SYSTEM LIFTER_MVCDL (* Lifter Control+Diagnostics with Feed & Takeoff Conveyors *)
  (* Standard: 61499-1; Classification: Simulation; ApplicationDomain: Assembly; Type: Dual Stroke Cylinder *)
  (* Version 0.5, 2008-02-18, JHC, Holobloc Inc, Added init delay to DIAGNOSTICS.LOG *)
  (* Version 0.4, 2007-11-08, JHC, Holobloc Inc, Changed device order: DIAGNOSTICS, MODEL, CONTROL. *)
  (* Version 0.3, 2007-07-08, JHC, Holobloc Inc, Added MODEL.CLOCK.CLK_DLY. *)
  (* Version 0.2, 2004-12-19, JHC, Rockwell Automation, Adjusted frame heights for WinXP. *)
  (* Version 0.1, 2004-11-12, JHC, Rockwell Automation, Combined XFER_MDL+FLT_MDL as in LIFTER_MVCL. *)
  (* Version 0.0, 2004-11-10, JHC, Rockwell Automation, Extended from LIFTER_MVCL. *)
  DEVICE DIAGNOSTICS : FRAME_DEVICE(BOUNDS := [100,360,485,150], GRID := [1,1])
    RESOURCE LOG : PANEL_RESOURCE(ROWS := 1, COLS := 1)
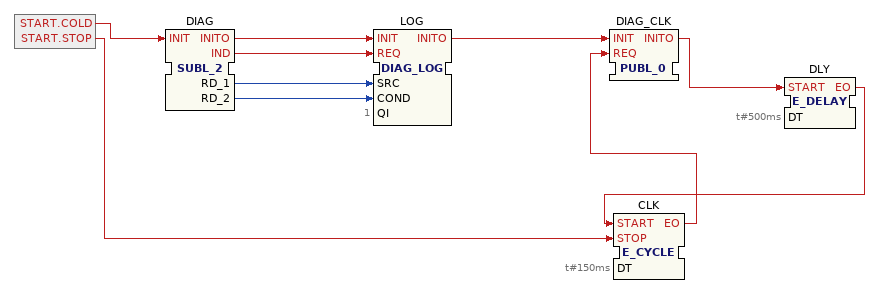
      FBS
        DIAG : SUBL_2;
        LOG : DIAG_LOG(QI := 1);
        CLK : E_CYCLE(DT := t#150ms);
        DIAG_CLK : PUBL_0;
        DLY : E_DELAY(DT := t#500ms);
      END_FBS
      EVENT_CONNECTIONS
        START.COLD TO DIAG.INIT;
        DIAG.INITO TO LOG.INIT;
        DIAG.IND TO LOG.REQ;
        LOG.INITO TO DIAG_CLK.INIT;
        CLK.EO TO DIAG_CLK.REQ;
        DIAG_CLK.INITO TO DLY.START;
        DLY.EO TO CLK.START;
        START.STOP TO CLK.STOP;
      END_CONNECTIONS
      DATA_CONNECTIONS
        DIAG.RD_1 TO LOG.SRC;
        DIAG.RD_2 TO LOG.COND;
      END_CONNECTIONS
    END_RESOURCE
    RESOURCE MONITOR : EMB_RES
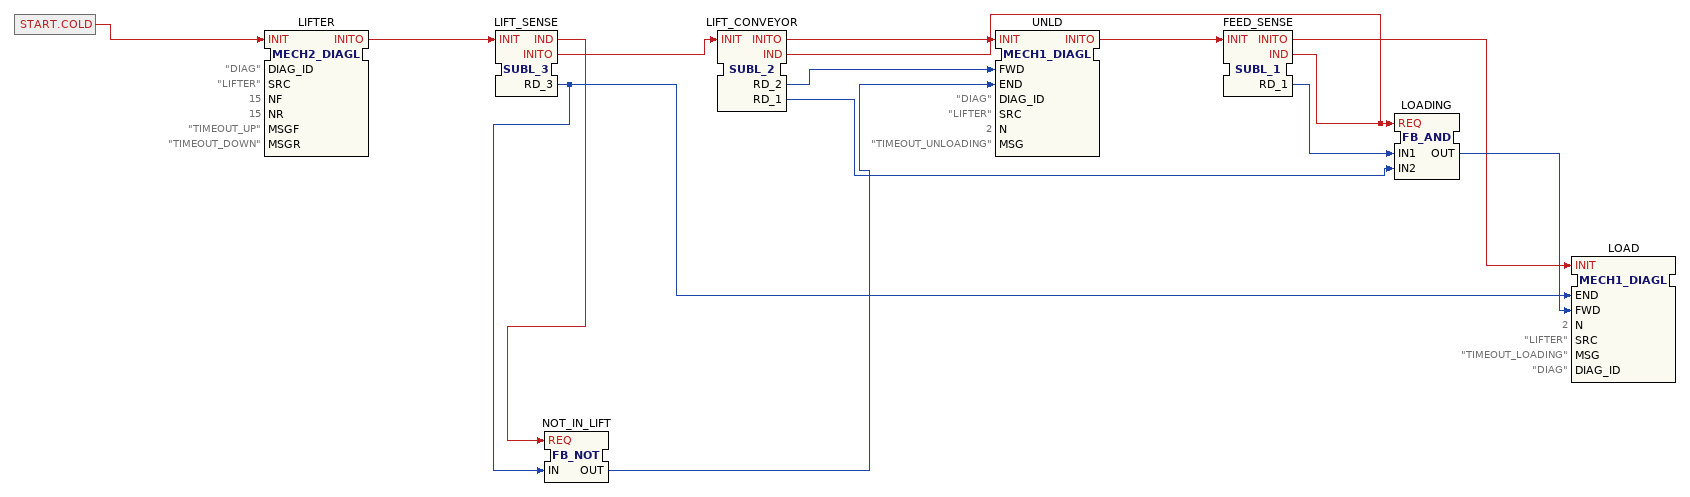
      FBS
        LIFTER : MECH2_DIAGL(DIAG_ID := "DIAG", SRC := "LIFTER", NF := 15, NR := 15, MSGF := "TIMEOUT_UP", MSGR := "TIMEOUT_DOWN");
        UNLD : MECH1_DIAGL(DIAG_ID := "DIAG", SRC := "LIFTER", N := 2, MSG := "TIMEOUT_UNLOADING"); (* Monitor Lift Unloading *)
        LIFT_CONVEYOR : SUBL_2;
        LIFT_SENSE : SUBL_3;
        NOT_IN_LIFT : FB_NOT;
        LOAD : MECH1_DIAGL(N := 2, SRC := "LIFTER", MSG := "TIMEOUT_LOADING", DIAG_ID := "DIAG");
        FEED_SENSE : SUBL_1;
        LOADING : FB_AND;
      END_FBS
      EVENT_CONNECTIONS
        START.COLD TO LIFTER.INIT;
        LIFT_SENSE.IND TO NOT_IN_LIFT.REQ;
        LIFTER.INITO TO LIFT_SENSE.INIT;
        LIFT_SENSE.INITO TO LIFT_CONVEYOR.INIT;
        LIFT_CONVEYOR.INITO TO UNLD.INIT;
        UNLD.INITO TO FEED_SENSE.INIT;
        FEED_SENSE.INITO TO LOAD.INIT;
        FEED_SENSE.IND TO LOADING.REQ;
        LIFT_CONVEYOR.IND TO LOADING.REQ;
      END_CONNECTIONS
      DATA_CONNECTIONS
        LIFT_CONVEYOR.RD_2 TO UNLD.FWD;
        NOT_IN_LIFT.OUT TO UNLD.END;
        LIFT_SENSE.RD_3 TO NOT_IN_LIFT.IN;
        LIFT_SENSE.RD_3 TO LOAD.END;
        LOADING.OUT TO LOAD.FWD;
        FEED_SENSE.RD_1 TO LOADING.IN1;
        LIFT_CONVEYOR.RD_1 TO LOADING.IN2;
      END_CONNECTIONS
    END_RESOURCE
  END_DEVICE
  DEVICE MODEL : FRAME_DEVICE(BOUNDS := [425,100,160,260])
    RESOURCE CLOCK : EMB_RES
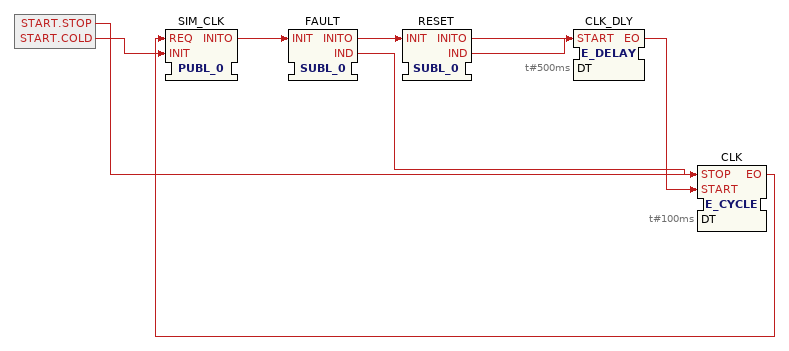
      FBS
        CLK : E_CYCLE(DT := t#100ms);
        SIM_CLK : PUBL_0;
        FAULT : SUBL_0;
        RESET : SUBL_0;
        CLK_DLY : E_DELAY(DT := t#500ms);
      END_FBS
      EVENT_CONNECTIONS
        START.STOP TO CLK.STOP;
        CLK.EO TO SIM_CLK.REQ;
        START.COLD TO SIM_CLK.INIT;
        SIM_CLK.INITO TO FAULT.INIT;
        FAULT.INITO TO RESET.INIT;
        FAULT.IND TO CLK.STOP;
        RESET.INITO TO CLK_DLY.START;
        RESET.IND TO CLK_DLY.START;
        CLK_DLY.EO TO CLK.START;
      END_CONNECTIONS
    END_RESOURCE
    RESOURCE FEED_MDL : EMB_RES
      FBS
        FEED : CNVG_MDLL(VF := 20, VS := 50);
        FEED_UNLD : SUBL_0;
        RESET : SUBL_0;
        WARN : SUBL_2;
        WARNING : LOADLE(LPOS := 100, STYLE := VSTYLE#PALLET, WKPC := [255,255,0], ID := "FEED_LOAD");
        JAM_OR_HALFIN : FB_OR;
        FAULT : SUBL_2;
        CRUSHED : E_PERMIT;
        DROPPED : LOADLE(ID := "FEED_LOAD", LPOS := 100, STYLE := VSTYLE#PALLET, WKPC := [255,0,0]);
      END_FBS
      EVENT_CONNECTIONS
        START.COLD TO FEED.INIT;
        FEED.INITO TO FEED_UNLD.INIT;
        FEED_UNLD.IND TO FEED.UNLD;
        FEED_UNLD.INITO TO RESET.INIT;
        RESET.IND TO FEED.UNLD;
        RESET.INITO TO WARN.INIT;
        START.COLD TO FAULT.INIT;
        WARN.INITO TO WARNING.INIT;
        JAM_OR_HALFIN.CNF TO WARNING.REQ;
        FAULT.IND TO CRUSHED.EI;
        CRUSHED.EO TO FEED.UNLD;
        FAULT.IND TO DROPPED.REQ;
        WARNING.INITO TO DROPPED.INIT;
        WARN.IND TO JAM_OR_HALFIN.REQ;
      END_CONNECTIONS
      DATA_CONNECTIONS
        WARN.RD_1 TO JAM_OR_HALFIN.IN1;
        WARN.RD_2 TO JAM_OR_HALFIN.IN2;
        JAM_OR_HALFIN.OUT TO WARNING.QI;
        FAULT.RD_1 TO CRUSHED.PERMIT;
        FAULT.RD_2 TO DROPPED.QI;
      END_CONNECTIONS
    END_RESOURCE
    RESOURCE LIFTER_MDL : EMB_RES
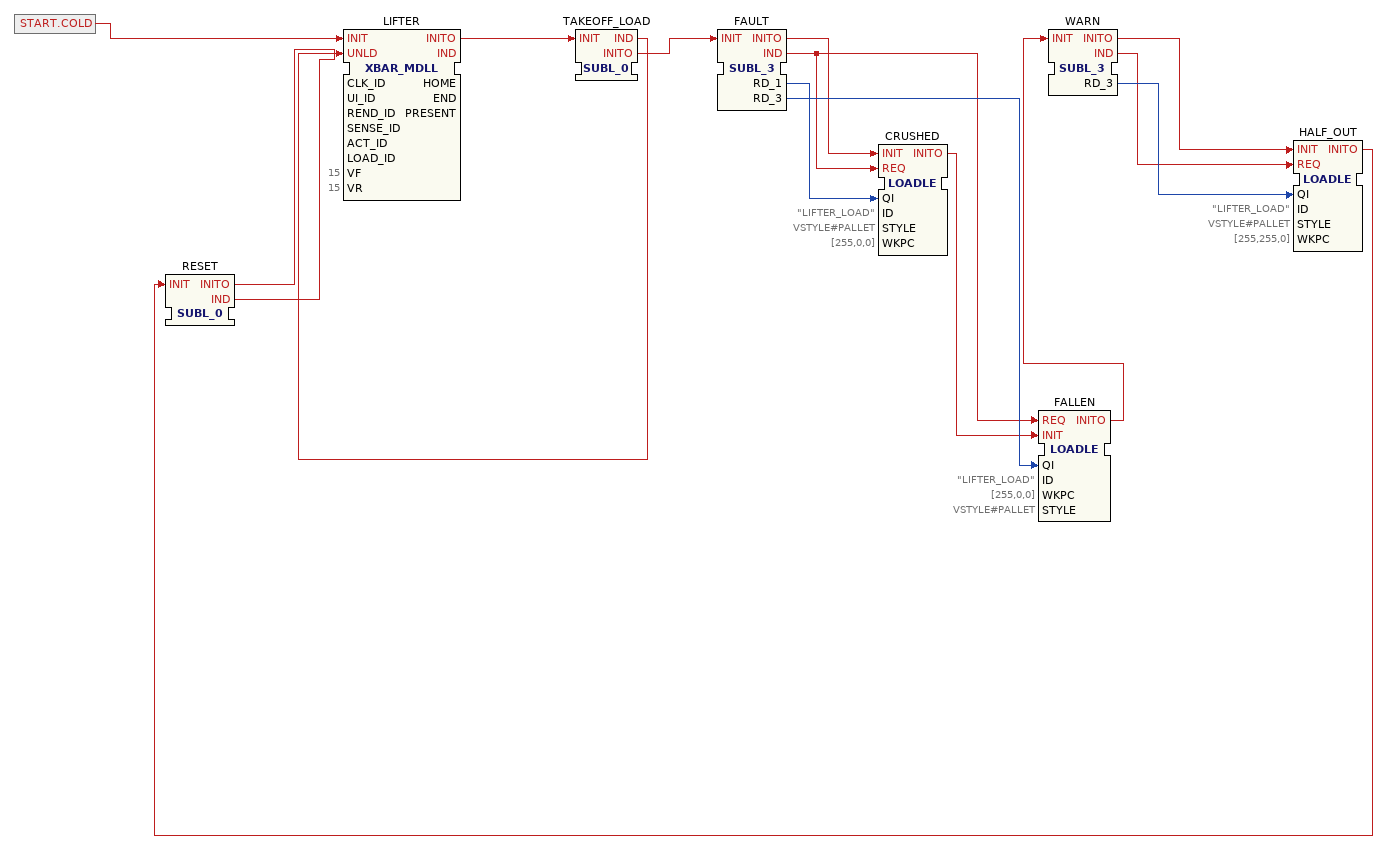
      FBS
        LIFTER : XBAR_MDLL(VF := 15, VR := 15);
        TAKEOFF_LOAD : SUBL_0;
        FAULT : SUBL_3;
        CRUSHED : LOADLE(ID := "LIFTER_LOAD", STYLE := VSTYLE#PALLET, WKPC := [255,0,0]);
        FALLEN : LOADLE(ID := "LIFTER_LOAD", WKPC := [255,0,0], STYLE := VSTYLE#PALLET);
        RESET : SUBL_0;
        WARN : SUBL_3;
        HALF_OUT : LOADLE(ID := "LIFTER_LOAD", STYLE := VSTYLE#PALLET, WKPC := [255,255,0]);
      END_FBS
      EVENT_CONNECTIONS
        START.COLD TO LIFTER.INIT;
        LIFTER.INITO TO TAKEOFF_LOAD.INIT;
        TAKEOFF_LOAD.IND TO LIFTER.UNLD;
        TAKEOFF_LOAD.INITO TO FAULT.INIT;
        FAULT.INITO TO CRUSHED.INIT;
        FAULT.IND TO CRUSHED.REQ;
        FAULT.IND TO FALLEN.REQ;
        CRUSHED.INITO TO FALLEN.INIT;
        WARN.INITO TO HALF_OUT.INIT;
        WARN.IND TO HALF_OUT.REQ;
        RESET.INITO TO LIFTER.UNLD;
        RESET.IND TO LIFTER.UNLD;
        FALLEN.INITO TO WARN.INIT;
        HALF_OUT.INITO TO RESET.INIT;
      END_CONNECTIONS
      DATA_CONNECTIONS
        FAULT.RD_1 TO CRUSHED.QI;
        FAULT.RD_3 TO FALLEN.QI;
        WARN.RD_3 TO HALF_OUT.QI;
      END_CONNECTIONS
    END_RESOURCE
    RESOURCE XFER_MDL : EMB_RES (* Pallet Transfer Model *)
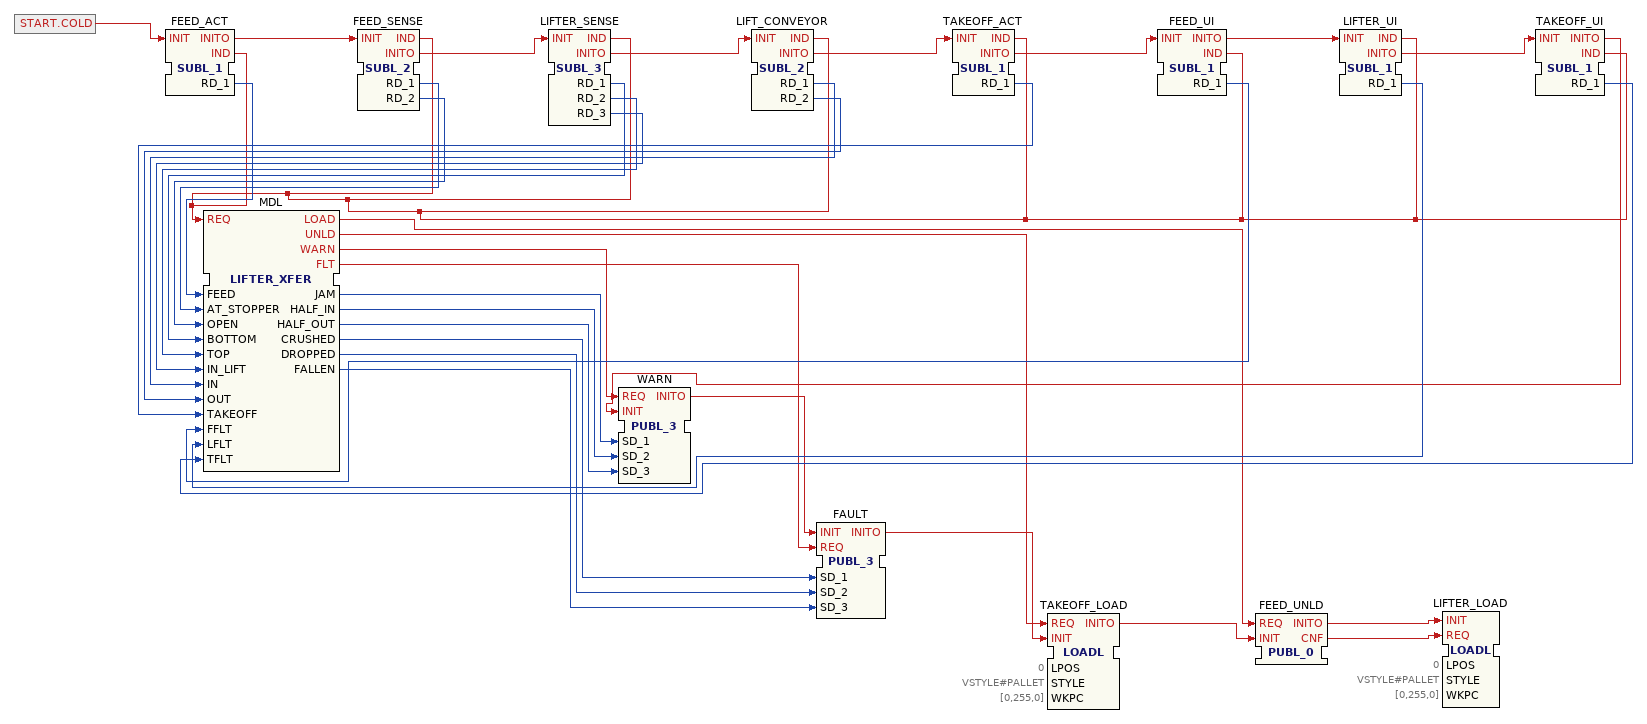
      FBS
        MDL : LIFTER_XFER;
        FEED_ACT : SUBL_1;
        FEED_SENSE : SUBL_2;
        LIFTER_SENSE : SUBL_3;
        LIFT_CONVEYOR : SUBL_2;
        TAKEOFF_ACT : SUBL_1;
        LIFTER_LOAD : LOADL(LPOS := 0, STYLE := VSTYLE#PALLET, WKPC := [0,255,0]);
        TAKEOFF_LOAD : LOADL(LPOS := 0, STYLE := VSTYLE#PALLET, WKPC := [0,255,0]);
        LIFTER_UI : SUBL_1;
        WARN : PUBL_3;
        FAULT : PUBL_3;
        FEED_UNLD : PUBL_0;
        FEED_UI : SUBL_1;
        TAKEOFF_UI : SUBL_1;
      END_FBS
      EVENT_CONNECTIONS
        START.COLD TO FEED_ACT.INIT;
        FEED_ACT.INITO TO FEED_SENSE.INIT;
        FEED_ACT.IND TO MDL.REQ;
        FEED_SENSE.IND TO MDL.REQ;
        FEED_SENSE.INITO TO LIFTER_SENSE.INIT;
        LIFTER_SENSE.IND TO MDL.REQ;
        LIFTER_SENSE.INITO TO LIFT_CONVEYOR.INIT;
        LIFT_CONVEYOR.IND TO MDL.REQ;
        LIFT_CONVEYOR.INITO TO TAKEOFF_ACT.INIT;
        TAKEOFF_ACT.IND TO MDL.REQ;
        LIFTER_UI.IND TO MDL.REQ;
        MDL.UNLD TO TAKEOFF_LOAD.REQ;
        WARN.INITO TO FAULT.INIT;
        MDL.WARN TO WARN.REQ;
        MDL.FLT TO FAULT.REQ;
        FAULT.INITO TO TAKEOFF_LOAD.INIT;
        MDL.LOAD TO FEED_UNLD.REQ;
        FEED_UNLD.INITO TO LIFTER_LOAD.INIT;
        FEED_UNLD.CNF TO LIFTER_LOAD.REQ;
        TAKEOFF_LOAD.INITO TO FEED_UNLD.INIT;
        TAKEOFF_ACT.INITO TO FEED_UI.INIT;
        FEED_UI.INITO TO LIFTER_UI.INIT;
        LIFTER_UI.INITO TO TAKEOFF_UI.INIT;
        TAKEOFF_UI.INITO TO WARN.INIT;
        FEED_UI.IND TO MDL.REQ;
        TAKEOFF_UI.IND TO MDL.REQ;
      END_CONNECTIONS
      DATA_CONNECTIONS
        FEED_ACT.RD_1 TO MDL.FEED;
        FEED_SENSE.RD_1 TO MDL.AT_STOPPER;
        LIFTER_SENSE.RD_1 TO MDL.BOTTOM;
        LIFTER_SENSE.RD_2 TO MDL.TOP;
        LIFTER_SENSE.RD_3 TO MDL.IN_LIFT;
        LIFT_CONVEYOR.RD_1 TO MDL.IN;
        LIFT_CONVEYOR.RD_2 TO MDL.OUT;
        TAKEOFF_ACT.RD_1 TO MDL.TAKEOFF;
        FEED_SENSE.RD_2 TO MDL.OPEN;
        LIFTER_UI.RD_1 TO MDL.LFLT;
        MDL.JAM TO WARN.SD_1;
        MDL.HALF_IN TO WARN.SD_2;
        MDL.HALF_OUT TO WARN.SD_3;
        MDL.CRUSHED TO FAULT.SD_1;
        MDL.DROPPED TO FAULT.SD_2;
        MDL.FALLEN TO FAULT.SD_3;
        FEED_UI.RD_1 TO MDL.FFLT;
        TAKEOFF_UI.RD_1 TO MDL.TFLT;
      END_CONNECTIONS
    END_RESOURCE
    RESOURCE TAKEOFF_MDL : EMB_RES
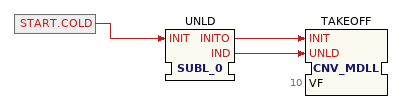
      FBS
        TAKEOFF : CNV_MDLL(VF := 10);
        UNLD : SUBL_0;
      END_FBS
      EVENT_CONNECTIONS
        START.COLD TO UNLD.INIT;
        UNLD.INITO TO TAKEOFF.INIT;
        UNLD.IND TO TAKEOFF.UNLD;
      END_CONNECTIONS
    END_RESOURCE
    RESOURCE UI : PANEL_RESOURCE(ROWS := 2, COLS := 2)
      FBS
        FAULT_IND : OUT_BOOL(LABEL := "FAULT ", C1 := [255,0,0]);
        RESET_PB : IN_EVENT(LABEL := "RESET");
        RESET : PUBL_0;
        LOAD_PB : IN_EVENT(LABEL := "LOAD");
        UNLD_PB : IN_EVENT(LABEL := "UNLOAD");
        FEED_LOAD : LOADL(STYLE := VSTYLE#PALLET, WKPC := [0,255,0]);
        UNLD : PUBL_0;
        FLT : E_RS;
        FAULT : SUBL_0;
      END_FBS
      EVENT_CONNECTIONS
        FAULT_IND.INITO TO RESET_PB.INIT;
        RESET_PB.INITO TO RESET.INIT;
        RESET_PB.IND TO RESET.REQ;
        START.COLD TO LOAD_PB.INIT;
        LOAD_PB.INITO TO FEED_LOAD.INIT;
        FEED_LOAD.INITO TO UNLD_PB.INIT;
        LOAD_PB.IND TO FEED_LOAD.REQ;
        UNLD_PB.INITO TO UNLD.INIT;
        UNLD_PB.IND TO UNLD.REQ;
        UNLD.INITO TO FAULT_IND.INIT;
        RESET.CNF TO UNLD.REQ;
        FLT.EO TO FAULT_IND.REQ;
        RESET.INITO TO FAULT.INIT;
        FAULT.IND TO FLT.S;
        UNLD.CNF TO FLT.R;
      END_CONNECTIONS
      DATA_CONNECTIONS
        FLT.Q TO FAULT_IND.IN;
      END_CONNECTIONS
    END_RESOURCE
    RESOURCE VIEW : VIEW_PANEL(DIA := 30, SIZE := [5,5], VERTICAL := 1)
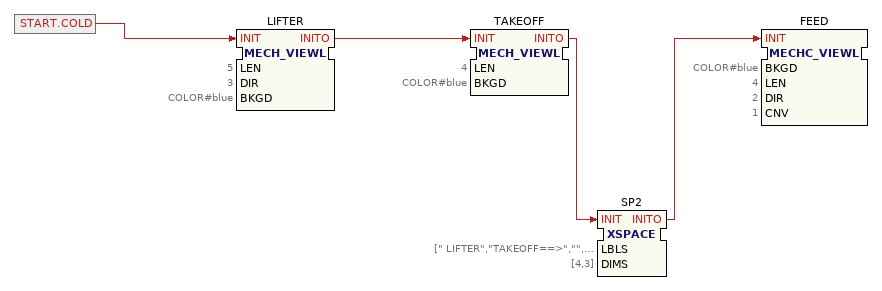
      FBS
        LIFTER : MECH_VIEWL(LEN := 5, DIR := 3, BKGD := COLOR#blue);
        FEED : MECHC_VIEWL(BKGD := COLOR#blue, LEN := 4, DIR := 2, CNV := 1); (* Feed Conveyor *)
        SP2 : XSPACE(LBLS := [" LIFTER","TAKEOFF==>","","<==FEED"], DIMS := [4,3]);
        TAKEOFF : MECH_VIEWL(LEN := 4, BKGD := COLOR#blue); (* Takeoff Conveyor *)
      END_FBS
      EVENT_CONNECTIONS
        TAKEOFF.INITO TO SP2.INIT;
        SP2.INITO TO FEED.INIT;
        START.COLD TO LIFTER.INIT;
        LIFTER.INITO TO TAKEOFF.INIT;
      END_CONNECTIONS
    END_RESOURCE
  END_DEVICE
  DEVICE CONTROL : FRAME_DEVICE(BOUNDS := [100,100,325,260], GRID := [3,2]) (* Lifter Control + HMI *)
    RESOURCE CTL : EMB_RES
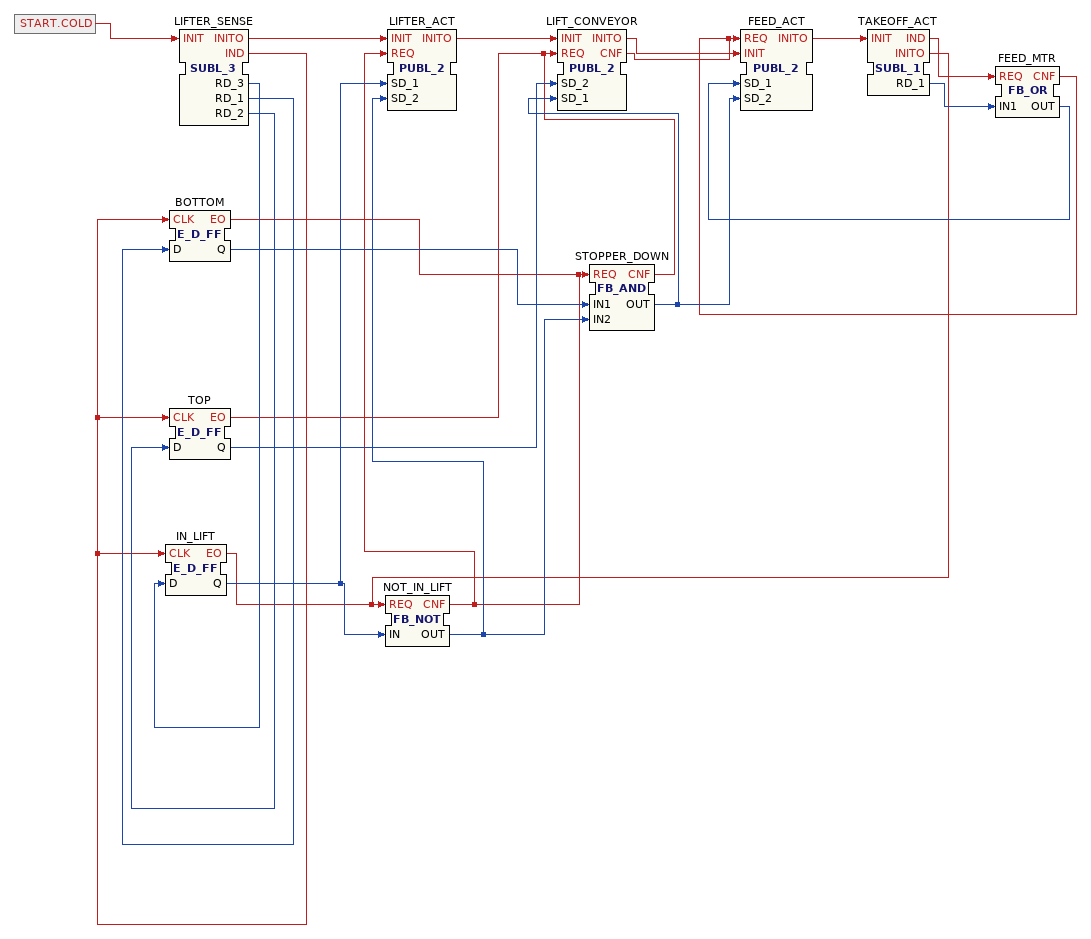
      FBS
        LIFTER_SENSE : SUBL_3;
        FEED_ACT : PUBL_2;
        LIFTER_ACT : PUBL_2;
        LIFT_CONVEYOR : PUBL_2;
        TAKEOFF_ACT : SUBL_1;
        FEED_MTR : FB_OR;
        IN_LIFT : E_D_FF;
        BOTTOM : E_D_FF;
        TOP : E_D_FF;
        NOT_IN_LIFT : FB_NOT;
        STOPPER_DOWN : FB_AND;
      END_FBS
      EVENT_CONNECTIONS
        START.COLD TO LIFTER_SENSE.INIT;
        FEED_ACT.INITO TO TAKEOFF_ACT.INIT;
        TAKEOFF_ACT.IND TO FEED_MTR.REQ;
        FEED_MTR.CNF TO FEED_ACT.REQ;
        LIFTER_SENSE.INITO TO LIFTER_ACT.INIT;
        LIFTER_ACT.INITO TO LIFT_CONVEYOR.INIT;
        LIFT_CONVEYOR.INITO TO FEED_ACT.INIT;
        LIFTER_SENSE.IND TO IN_LIFT.CLK;
        LIFTER_SENSE.IND TO TOP.CLK;
        LIFTER_SENSE.IND TO BOTTOM.CLK;
        IN_LIFT.EO TO NOT_IN_LIFT.REQ;
        NOT_IN_LIFT.CNF TO LIFTER_ACT.REQ;
        TOP.EO TO LIFT_CONVEYOR.REQ;
        BOTTOM.EO TO STOPPER_DOWN.REQ;
        NOT_IN_LIFT.CNF TO STOPPER_DOWN.REQ;
        TAKEOFF_ACT.INITO TO NOT_IN_LIFT.REQ;
        LIFT_CONVEYOR.CNF TO FEED_ACT.REQ;
        STOPPER_DOWN.CNF TO LIFT_CONVEYOR.REQ;
      END_CONNECTIONS
      DATA_CONNECTIONS
        TAKEOFF_ACT.RD_1 TO FEED_MTR.IN1;
        FEED_MTR.OUT TO FEED_ACT.SD_1;
        LIFTER_SENSE.RD_3 TO IN_LIFT.D;
        LIFTER_SENSE.RD_1 TO BOTTOM.D;
        LIFTER_SENSE.RD_2 TO TOP.D;
        IN_LIFT.Q TO NOT_IN_LIFT.IN;
        IN_LIFT.Q TO LIFTER_ACT.SD_1;
        NOT_IN_LIFT.OUT TO LIFTER_ACT.SD_2;
        TOP.Q TO LIFT_CONVEYOR.SD_2;
        BOTTOM.Q TO STOPPER_DOWN.IN1;
        NOT_IN_LIFT.OUT TO STOPPER_DOWN.IN2;
        STOPPER_DOWN.OUT TO FEED_ACT.SD_2;
        STOPPER_DOWN.OUT TO LIFT_CONVEYOR.SD_1;
      END_CONNECTIONS
    END_RESOURCE
    RESOURCE TAKEOFF_SENSORS : PANEL_RESOURCE(ROWS := 2, COLS := 1)
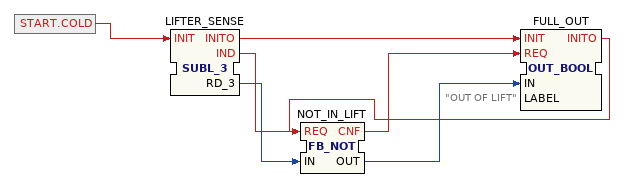
      FBS
        LIFTER_SENSE : SUBL_3;
        FULL_OUT : OUT_BOOL(LABEL := "OUT OF LIFT");
        NOT_IN_LIFT : FB_NOT;
      END_FBS
      EVENT_CONNECTIONS
        START.COLD TO LIFTER_SENSE.INIT;
        LIFTER_SENSE.INITO TO FULL_OUT.INIT;
        LIFTER_SENSE.IND TO NOT_IN_LIFT.REQ;
        NOT_IN_LIFT.CNF TO FULL_OUT.REQ;
        FULL_OUT.INITO TO NOT_IN_LIFT.REQ;
      END_CONNECTIONS
      DATA_CONNECTIONS
        LIFTER_SENSE.RD_3 TO NOT_IN_LIFT.IN;
        NOT_IN_LIFT.OUT TO FULL_OUT.IN;
      END_CONNECTIONS
    END_RESOURCE
    RESOURCE TAKEOFF_ACTUATORS : PANEL_RESOURCE
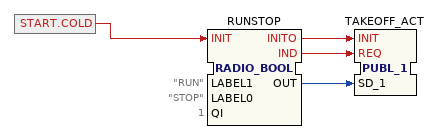
      FBS
        TAKEOFF_ACT : PUBL_1;
        RUNSTOP : RADIO_BOOL(LABEL1 := "RUN", LABEL0 := "STOP", QI := 1);
      END_FBS
      EVENT_CONNECTIONS
        START.COLD TO RUNSTOP.INIT;
        RUNSTOP.INITO TO TAKEOFF_ACT.INIT;
        RUNSTOP.IND TO TAKEOFF_ACT.REQ;
      END_CONNECTIONS
      DATA_CONNECTIONS
        RUNSTOP.OUT TO TAKEOFF_ACT.SD_1;
      END_CONNECTIONS
    END_RESOURCE
    RESOURCE LIFT_SENSORS : PANEL_RESOURCE(ROWS := 2, COLS := 2)
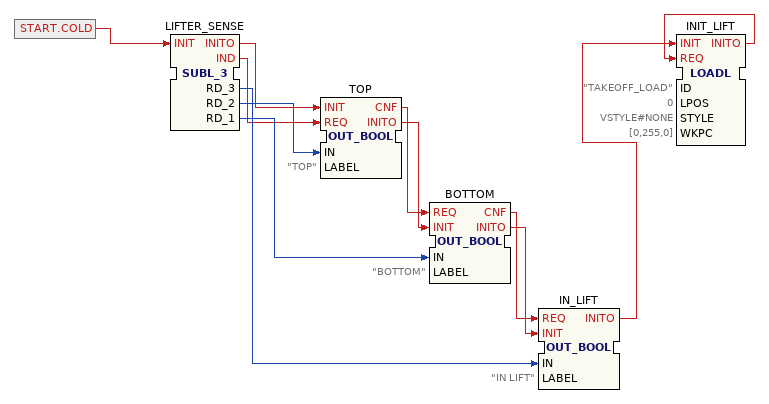
      FBS
        LIFTER_SENSE : SUBL_3;
        IN_LIFT : OUT_BOOL(LABEL := "IN LIFT");
        TOP : OUT_BOOL(LABEL := "TOP");
        BOTTOM : OUT_BOOL(LABEL := "BOTTOM");
        INIT_LIFT : LOADL(ID := "TAKEOFF_LOAD", LPOS := 0, STYLE := VSTYLE#NONE, WKPC := [0,255,0]);
      END_FBS
      EVENT_CONNECTIONS
        START.COLD TO LIFTER_SENSE.INIT;
        TOP.CNF TO BOTTOM.REQ;
        TOP.INITO TO BOTTOM.INIT;
        LIFTER_SENSE.INITO TO TOP.INIT;
        LIFTER_SENSE.IND TO TOP.REQ;
        BOTTOM.CNF TO IN_LIFT.REQ;
        BOTTOM.INITO TO IN_LIFT.INIT;
        IN_LIFT.INITO TO INIT_LIFT.INIT;
        INIT_LIFT.INITO TO INIT_LIFT.REQ;
      END_CONNECTIONS
      DATA_CONNECTIONS
        LIFTER_SENSE.RD_3 TO IN_LIFT.IN;
        LIFTER_SENSE.RD_2 TO TOP.IN;
        LIFTER_SENSE.RD_1 TO BOTTOM.IN;
      END_CONNECTIONS
    END_RESOURCE
    RESOURCE LIFT_ACTUATORS : PANEL_RESOURCE(ROWS := 2, COLS := 2)
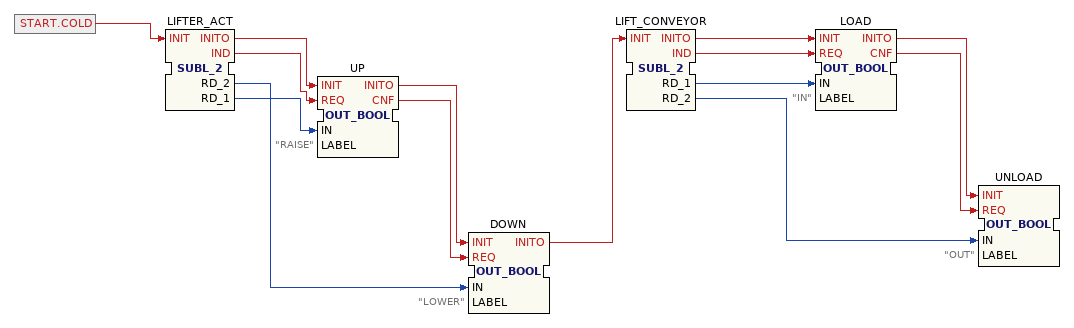
      FBS
        UP : OUT_BOOL(LABEL := "RAISE");
        LIFTER_ACT : SUBL_2;
        DOWN : OUT_BOOL(LABEL := "LOWER");
        LOAD : OUT_BOOL(LABEL := "IN");
        UNLOAD : OUT_BOOL(LABEL := "OUT");
        LIFT_CONVEYOR : SUBL_2;
      END_FBS
      EVENT_CONNECTIONS
        START.COLD TO LIFTER_ACT.INIT;
        LIFTER_ACT.INITO TO UP.INIT;
        UP.INITO TO DOWN.INIT;
        LIFTER_ACT.IND TO UP.REQ;
        UP.CNF TO DOWN.REQ;
        DOWN.INITO TO LIFT_CONVEYOR.INIT;
        LIFT_CONVEYOR.INITO TO LOAD.INIT;
        LOAD.INITO TO UNLOAD.INIT;
        LOAD.CNF TO UNLOAD.REQ;
        LIFT_CONVEYOR.IND TO LOAD.REQ;
      END_CONNECTIONS
      DATA_CONNECTIONS
        LIFTER_ACT.RD_2 TO DOWN.IN;
        LIFTER_ACT.RD_1 TO UP.IN;
        LIFT_CONVEYOR.RD_1 TO LOAD.IN;
        LIFT_CONVEYOR.RD_2 TO UNLOAD.IN;
      END_CONNECTIONS
    END_RESOURCE
    RESOURCE FEED_SENSORS : PANEL_RESOURCE(ROWS := 2, COLS := 1)
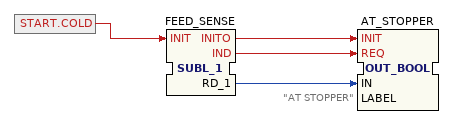
      FBS
        FEED_SENSE : SUBL_1;
        AT_STOPPER : OUT_BOOL(LABEL := "AT STOPPER");
      END_FBS
      EVENT_CONNECTIONS
        START.COLD TO FEED_SENSE.INIT;
        FEED_SENSE.INITO TO AT_STOPPER.INIT;
        FEED_SENSE.IND TO AT_STOPPER.REQ;
      END_CONNECTIONS
      DATA_CONNECTIONS
        FEED_SENSE.RD_1 TO AT_STOPPER.IN;
      END_CONNECTIONS
    END_RESOURCE
    RESOURCE FEED_ACTUATORS : PANEL_RESOURCE(ROWS := 2, COLS := 1)
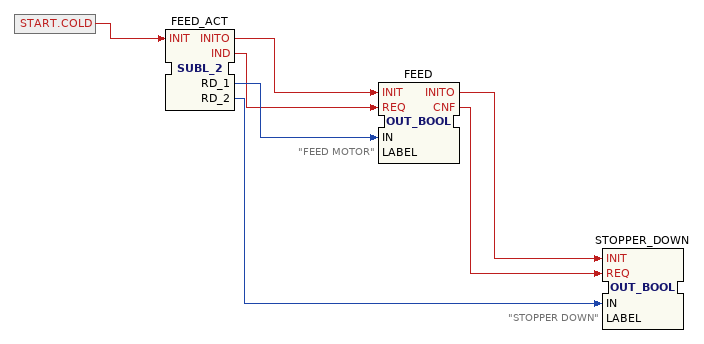
      FBS
        FEED : OUT_BOOL(LABEL := "FEED MOTOR");
        FEED_ACT : SUBL_2;
        STOPPER_DOWN : OUT_BOOL(LABEL := "STOPPER DOWN");
      END_FBS
      EVENT_CONNECTIONS
        START.COLD TO FEED_ACT.INIT;
        FEED_ACT.INITO TO FEED.INIT;
        FEED_ACT.IND TO FEED.REQ;
        FEED.INITO TO STOPPER_DOWN.INIT;
        FEED.CNF TO STOPPER_DOWN.REQ;
      END_CONNECTIONS
      DATA_CONNECTIONS
        FEED_ACT.RD_1 TO FEED.IN;
        FEED_ACT.RD_2 TO STOPPER_DOWN.IN;
      END_CONNECTIONS
    END_RESOURCE
  END_DEVICE
END_SYSTEM
